{attribute 'GeneratedUsingTerminal: EL6021-0000-0018'}
{attribute addProperty BoxType "EL6021-0000-0018"}
{attribute addProperty Id "COM_TxPDO_Map_InputsAT %I*COM_TxPDO_Map_Inputs_3801C95E30COM_RxPDO_Map_OutputsAT %Q*COM_RxPDO_Map_Outputs_DEF408EC27WcStateAT %I*WcState_9091E0EB2InfoDataAT %I*InfoData_94A18F5E2"}
{attribute addProperty CRC "4230424261"}
{attribute addProperty Size "61"}
TYPE EL6021_FC2726C5 EXTENDS EtcSlaveTerminalBase_947E5A46 :
STRUCT
	{attribute addProperty Name "COM_TxPDO_Map_Inputs"}
	COM_TxPDO_Map_Inputs : COM_TxPDO_Map_Inputs_3801C95E;
	{attribute addProperty Name "COM_RxPDO_Map_Outputs"}
	COM_RxPDO_Map_Outputs : COM_RxPDO_Map_Outputs_DEF408EC;
	{attribute addProperty Name "WcState"}
	WcState : WcState_9091E0EB;
	{attribute addProperty Name "InfoData"}
	InfoData : InfoData_94A18F5E;
END_STRUCT
END_TYPE

(* stored: Version 1.2.0.0, ProductVersion 3.1.4024.9
   DUT EL6021_FC2726C5: Id {97955b0a-0074-469f-bfa3-23366cc9e523} *)
